INTERFACE ITF_Updater

METHOD GetTypeID : BYTE
VAR_INPUT
END_VAR
END_METHOD

METHOD GetVersion : BYTE
VAR_INPUT
END_VAR
END_METHOD

METHOD SetSenderTimestamp : BOOL
VAR_INPUT
END_VAR
END_METHOD

METHOD SetTimeDifference : BOOL
VAR_INPUT
END_VAR
END_METHOD

METHOD TryApplyPayload : HRESULT
VAR_INPUT
	PacketAddress	: PVOID;
	PacketLength	: UINT;
	EspHost			: ITF_EspHost;
END_VAR
END_METHOD

METHOD TryGetContents : HRESULT
VAR_INPUT
	Host	: ITF_EspHost;
	Content	: REFERENCE TO STRING(1024);
END_VAR
END_METHOD

METHOD TrySendInstruction : HRESULT
VAR_INPUT
END_VAR
END_METHOD

END_INTERFACE

(* stored: Version 1.1.0.1
   Itf ITF_Updater: Id {55c350b8-68d9-436d-a671-afe1ee501105}
   Method GetTypeID: Id {b056be6e-1afa-4f32-b4a4-e1157d0ff783}
   Method GetVersion: Id {8abd07a8-5181-44f8-9e43-784834337c4c}
   Method SetSenderTimestamp: Id {7336ed7e-a0c5-4c6d-a463-70189b36404b}
   Method SetTimeDifference: Id {c905b475-5030-446d-b4ac-81e4f17b9636}
   Method TryApplyPayload: Id {62f62d39-4422-4e09-9635-584ba5e34fa0}
   Method TryGetContents: Id {4c68d0bc-3165-4bef-a0a5-d07117a57984}
   Method TrySendInstruction: Id {69d6b1b3-7d13-47d8-8d01-f870d18e7678} *)
